FUNCTION_BLOCK KlebeStation
VAR_INPUT
END_VAR
VAR_OUTPUT
END_VAR
VAR
END_VAR

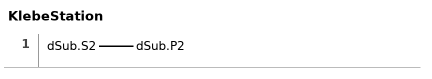
// NETWORK 1
dSub.P2 := dSub.S2;

END_FUNCTION_BLOCK

(* stored: Version 1.1.0.1, ProductVersion 3.1.4022.6
   POU KlebeStation: Id {89235d84-7b67-4ef3-9a17-571134cdcb1d}, SpecialFunc None *)
